// TIA Portal project "Giro de un motor trifasico NOT" (V17)

(* hardware
DEVICE "S7-1200 station_1"  S7-1200 Station
   slot 0: "Rack_0"  S7-1200 Rack  Rack  V1.0
   slot 1: "PLC_1"  CPU 1212C AC/DC/Rly  6ES7 212-1BE40-0XB0  V4.5
*)

// ===== PLC "PLC_1"  CPU 1212C AC/DC/Rly =====

VAR_GLOBAL   // PLC tag table "Default tag table"
   "Marcha" AT %I0.0 : Bool;
   "Paro" AT %I0.1 : Bool;
   "Led Verde" AT %Q0.0 : Bool;
   "Led Rojo" AT %Q0.1 : Bool;
   "Motor_Dcha" AT %Q0.2 : Bool;
   "B_Dcha" AT %I0.2 : Bool;
   "Motor_Dcha_Indic" AT %Q0.4 : Bool;
   "B_Izq" AT %I0.3 : Bool;
   "Motor_Izq" AT %Q0.3 : Bool;
   "Motor_Izq_Indic" AT %Q0.5 : Bool;
END_VAR

FUNCTION "MHJ-PLC-Lab-Function-S71200" : Void   // FC9000, SCL
{ S7_Optimized_Access := 'TRUE' }
VERSION : 0.1
   VAR_TEMP
      rdTimeReturn : Int;
      outputTime : DTL;
      SyncVal : Byte;
      forVal : Int;
      forVal_2 : Int;
      Value : Byte;
   END_VAR
   VAR CONSTANT
      CompVal : Byte := 16#34;
      Value_01 : Byte := 16#11;
      Value_01_DW : DWord := 16#A165_D992;
      Value_02_DW : DWord := 16#58BE_4401;
   END_VAR
BEGIN

   #Value:=PEEK(area := 16#82,
        dbNumber := 0,
        byteOffset := 511);
   #Value := #Value + 1;

   POKE(area := 16#82,
        dbNumber := 0,
        byteOffset := 511,
        value := #Value);

   POKE(area:=16#81,
        dbNumber:=0,
        byteOffset:=1016,
        value:=#Value_01_DW);
   POKE(area := 16#81,
        dbNumber := 0,
        byteOffset := 1020,
        value := #Value_02_DW);

   POKE(area := 16#81,
        dbNumber := 0,
        byteOffset := 511,
        value := B#16#00);

   FOR #forVal := 0 TO 120 DO
       FOR #forVal_2:=0 TO 10 DO
           #rdTimeReturn:=RD_SYS_T(#outputTime);
           #rdTimeReturn := WR_SYS_T(#outputTime);
           #rdTimeReturn := RD_SYS_T(#outputTime);
           #rdTimeReturn := WR_SYS_T(#outputTime);
       END_FOR;
       #SyncVal:= PEEK(area := 16#81,
                      dbNumber := 0,
                      byteOffset := 511);
       IF #SyncVal = #CompVal THEN
          GOTO M_1;
       END_IF;
   END_FOR;
   RETURN;

   M_1:
   POKE(area := 16#81,
        dbNumber := 0,
        byteOffset := 511,
        value := B#16#0);
END_FUNCTION

ORGANIZATION_BLOCK "Main"   // OB1, LAD, ProgramCycle
TITLE = "Main Program Sweep (Cycle)"
{ S7_Optimized_Access := 'TRUE' }
VERSION : 0.1
   VAR_INPUT
      Initial_Call : Bool;   // Initial call of this OB
      Remanence : Bool;   // =True, if remanent data are available
   END_VAR
BEGIN

REGION Network 1
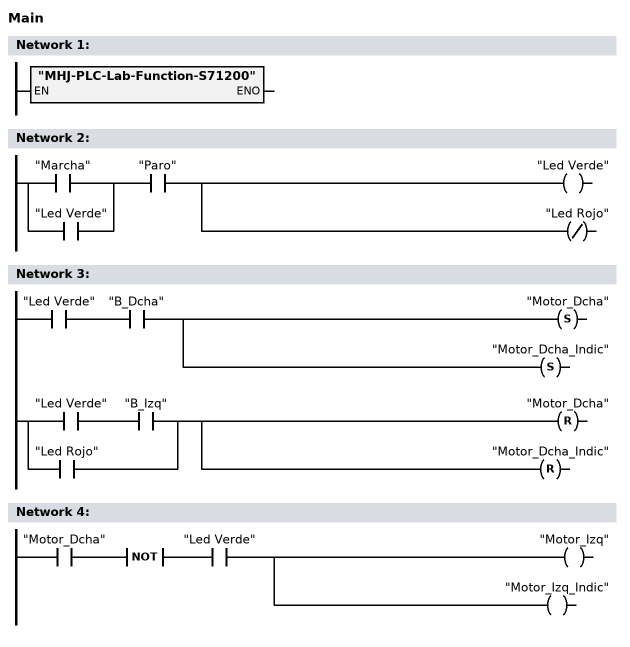
   RUNG wire#powerrail
      "MHJ-PLC-Lab-Function-S71200"()
   END_RUNG
   // the same network as SCL:
   "MHJ-PLC-Lab-Function-S71200"();
END_REGION

REGION Network 2
   RUNG wire#powerrail
      Contact( "Marcha" )
      wire#w1
      Contact( "Paro" )
      wire#w2
      Coil( "Led Verde" )
   END_RUNG
   RUNG wire#powerrail
      Contact( "Led Verde" )
   END_RUNG wire#w1
   RUNG wire#w2
      I_Coil( "Led Rojo" )
   END_RUNG
   // the same network as SCL:
   "Led Verde" := ("Marcha" OR "Led Verde") AND "Paro";
   "Led Rojo" := NOT "Led Verde";
END_REGION

REGION Network 3
   RUNG wire#powerrail
      Contact( "Led Verde" )
      Contact( "B_Dcha" )
      wire#w1
      S_Coil( "Motor_Dcha" )
   END_RUNG
   RUNG wire#w1
      S_Coil( "Motor_Dcha_Indic" )
   END_RUNG
   RUNG wire#powerrail
      Contact( "Led Verde" )
      Contact( "B_Izq" )
      wire#w2
      R_Coil( "Motor_Dcha" )
   END_RUNG
   RUNG wire#powerrail
      Contact( "Led Rojo" )
   END_RUNG wire#w2
   RUNG wire#w2
      R_Coil( "Motor_Dcha_Indic" )
   END_RUNG
   // the same network as SCL:
   IF "Led Verde" AND "B_Dcha" THEN
       "Motor_Dcha" := TRUE;
       "Motor_Dcha_Indic" := TRUE;
   END_IF;
   IF ("Led Verde" AND "B_Izq") OR "Led Rojo" THEN
       "Motor_Dcha" := FALSE;
       "Motor_Dcha_Indic" := FALSE;
   END_IF;
END_REGION

REGION Network 4
   RUNG wire#powerrail
      Contact( "Motor_Dcha" )
      Not()
      Contact( "Led Verde" )
      wire#w1
      Coil( "Motor_Izq" )
   END_RUNG
   RUNG wire#w1
      Coil( "Motor_Izq_Indic" )
   END_RUNG
   // the same network as SCL:
   "Motor_Izq" := NOT "Motor_Dcha" AND "Led Verde";
   "Motor_Izq_Indic" := "Motor_Izq";
END_REGION
END_ORGANIZATION_BLOCK